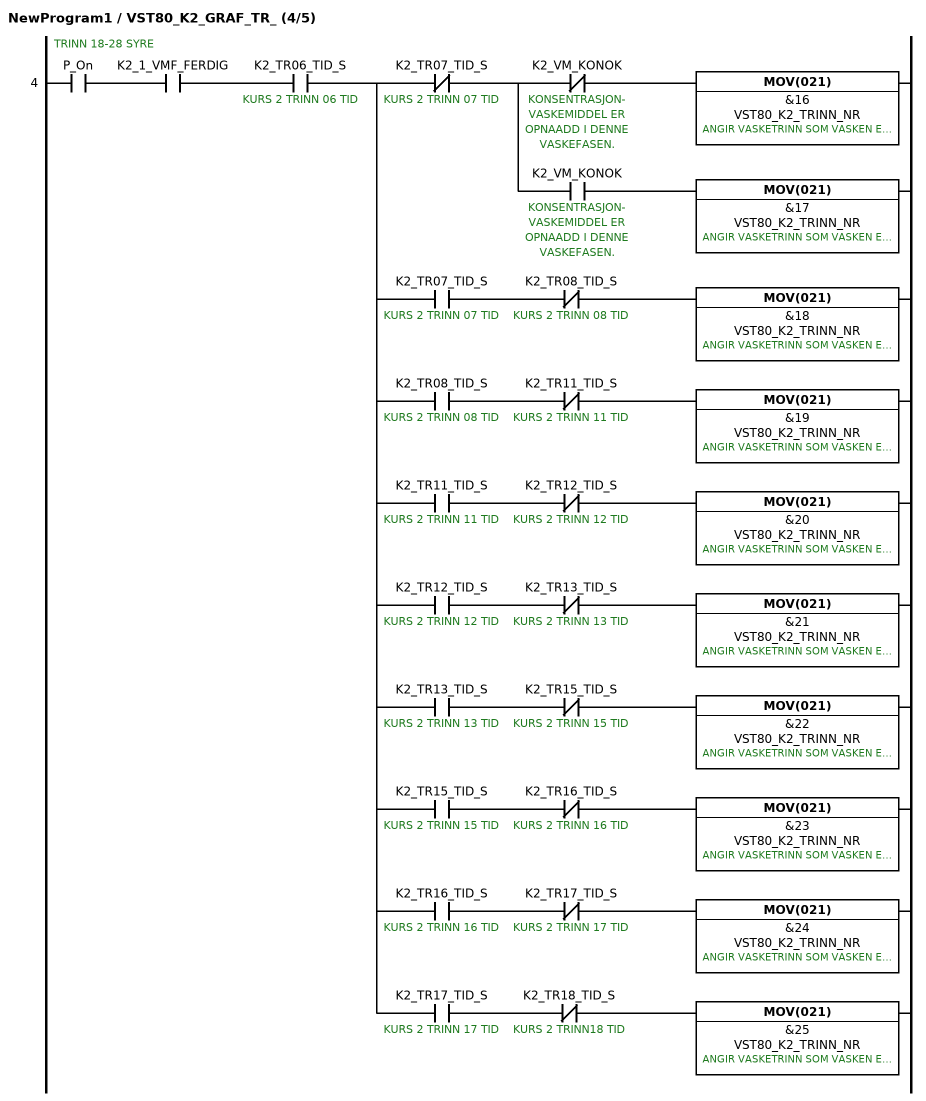
; [picture p264: NewProgram1 / VST80_K2_GRAF_TR_, rungs 4-4]
; rung 4: TRINN 18-28 SYRE
LD P_On
AND K2_1_VMF_FERDIG
AND K2_TR06_TID_S  ; KURS 2 TRINN 06 TID
OUT TR0
ANDNOT K2_TR07_TID_S  ; KURS 2 TRINN 07 TID
OUT TR1
ANDNOT K2_VM_KONOK  ; KONSENTRASJON-VASKEMIDDEL ER OPNAADD I DENNE VASKEFASEN.
MOV(021) &16 VST80_K2_TRINN_NR  ; ANGIR VASKETRINN SOM VASKEN ER I
LD TR1
AND K2_VM_KONOK  ; KONSENTRASJON-VASKEMIDDEL ER OPNAADD I DENNE VASKEFASEN.
MOV(021) &17 VST80_K2_TRINN_NR  ; ANGIR VASKETRINN SOM VASKEN ER I
LD TR0
AND K2_TR07_TID_S  ; KURS 2 TRINN 07 TID
ANDNOT K2_TR08_TID_S  ; KURS 2 TRINN 08 TID
MOV(021) &18 VST80_K2_TRINN_NR  ; ANGIR VASKETRINN SOM VASKEN ER I
LD TR0
AND K2_TR08_TID_S  ; KURS 2 TRINN 08 TID
ANDNOT K2_TR11_TID_S  ; KURS 2 TRINN 11 TID
MOV(021) &19 VST80_K2_TRINN_NR  ; ANGIR VASKETRINN SOM VASKEN ER I
LD TR0
AND K2_TR11_TID_S  ; KURS 2 TRINN 11 TID
ANDNOT K2_TR12_TID_S  ; KURS 2 TRINN 12 TID
MOV(021) &20 VST80_K2_TRINN_NR  ; ANGIR VASKETRINN SOM VASKEN ER I
LD TR0
AND K2_TR12_TID_S  ; KURS 2 TRINN 12 TID
ANDNOT K2_TR13_TID_S  ; KURS 2 TRINN 13 TID
MOV(021) &21 VST80_K2_TRINN_NR  ; ANGIR VASKETRINN SOM VASKEN ER I
LD TR0
AND K2_TR13_TID_S  ; KURS 2 TRINN 13 TID
ANDNOT K2_TR15_TID_S  ; KURS 2 TRINN 15 TID
MOV(021) &22 VST80_K2_TRINN_NR  ; ANGIR VASKETRINN SOM VASKEN ER I
LD TR0
AND K2_TR15_TID_S  ; KURS 2 TRINN 15 TID
ANDNOT K2_TR16_TID_S  ; KURS 2 TRINN 16 TID
MOV(021) &23 VST80_K2_TRINN_NR  ; ANGIR VASKETRINN SOM VASKEN ER I
LD TR0
AND K2_TR16_TID_S  ; KURS 2 TRINN 16 TID
ANDNOT K2_TR17_TID_S  ; KURS 2 TRINN 17 TID
MOV(021) &24 VST80_K2_TRINN_NR  ; ANGIR VASKETRINN SOM VASKEN ER I
LD TR0
AND K2_TR17_TID_S  ; KURS 2 TRINN 17 TID
ANDNOT K2_TR18_TID_S  ; KURS 2 TRINN18 TID
MOV(021) &25 VST80_K2_TRINN_NR  ; ANGIR VASKETRINN SOM VASKEN ER I

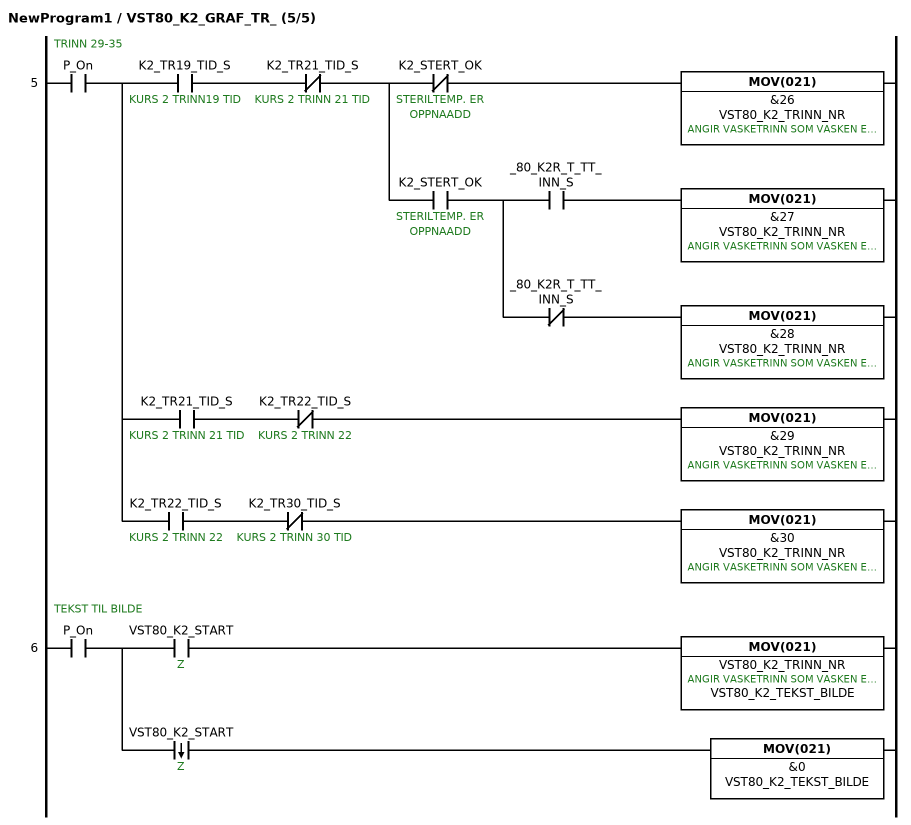
; rung 5: TRINN 29-35
LD P_On
OUT TR0
AND K2_TR19_TID_S  ; KURS 2 TRINN19 TID
ANDNOT K2_TR21_TID_S  ; KURS 2 TRINN 21 TID
OUT TR1
ANDNOT K2_STERT_OK  ; STERILTEMP. ER OPPNAADD
MOV(021) &26 VST80_K2_TRINN_NR  ; ANGIR VASKETRINN SOM VASKEN ER I
LD TR1
AND K2_STERT_OK  ; STERILTEMP. ER OPPNAADD
OUT TR1
AND _80_K2R_T_TT_INN_S
MOV(021) &27 VST80_K2_TRINN_NR  ; ANGIR VASKETRINN SOM VASKEN ER I
LD TR1
ANDNOT _80_K2R_T_TT_INN_S
MOV(021) &28 VST80_K2_TRINN_NR  ; ANGIR VASKETRINN SOM VASKEN ER I
LD TR0
AND K2_TR21_TID_S  ; KURS 2 TRINN 21 TID
ANDNOT K2_TR22_TID_S  ; KURS 2 TRINN 22
MOV(021) &29 VST80_K2_TRINN_NR  ; ANGIR VASKETRINN SOM VASKEN ER I
LD TR0
AND K2_TR22_TID_S  ; KURS 2 TRINN 22
ANDNOT K2_TR30_TID_S  ; KURS 2 TRINN 30 TID
MOV(021) &30 VST80_K2_TRINN_NR  ; ANGIR VASKETRINN SOM VASKEN ER I
; rung 6: TEKST TIL BILDE
LD P_On
OUT TR0
AND VST80_K2_START  ; Z
MOV(021) VST80_K2_TRINN_NR VST80_K2_TEKST_BILDE  ; ANGIR VASKETRINN SOM VASKEN ER I
LD TR0
%AND VST80_K2_START  ; Z
MOV(021) &0 VST80_K2_TEKST_BILDE
; rung 7: Ingen_kommentar_funnet

### Section VST80_K2_GRAF_FEIL_TXT

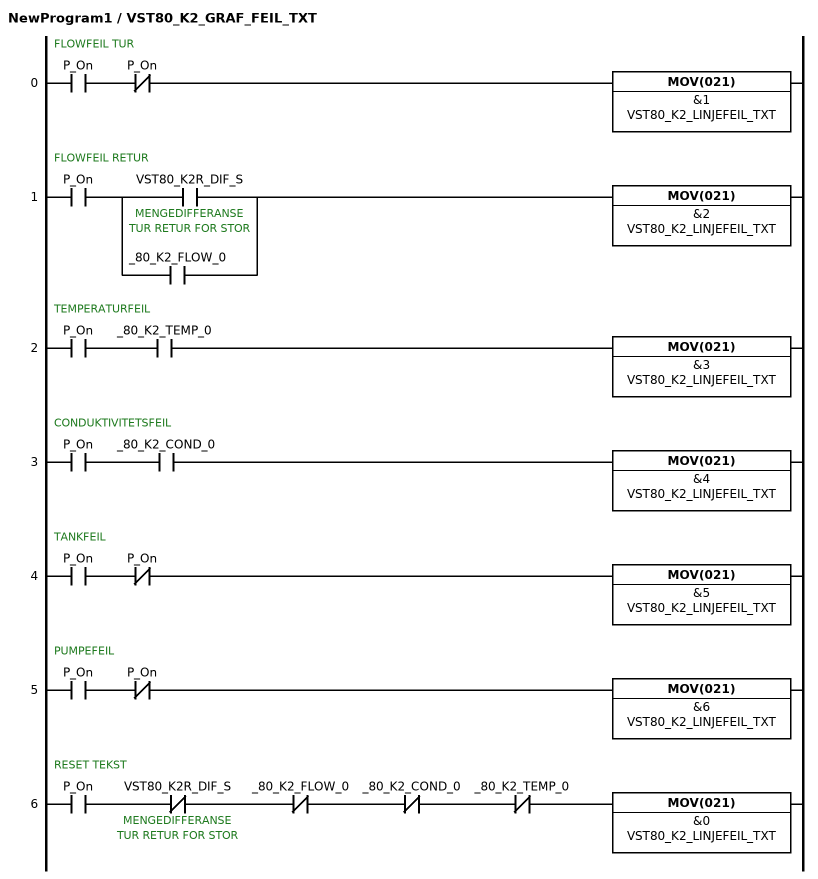
; rung 0: FLOWFEIL TUR
LD P_On
ANDNOT P_On
MOV(021) &1 VST80_K2_LINJEFEIL_TXT
; rung 1: FLOWFEIL RETUR
LD P_On
LD VST80_K2R_DIF_S  ; MENGEDIFFERANSE TUR RETUR FOR STOR
OR _80_K2_FLOW_0
ANDLD
MOV(021) &2 VST80_K2_LINJEFEIL_TXT
; rung 2: TEMPERATURFEIL
LD P_On
AND _80_K2_TEMP_0
MOV(021) &3 VST80_K2_LINJEFEIL_TXT
; rung 3: CONDUKTIVITETSFEIL
LD P_On
AND _80_K2_COND_0
MOV(021) &4 VST80_K2_LINJEFEIL_TXT
; rung 4: TANKFEIL
LD P_On
ANDNOT P_On
MOV(021) &5 VST80_K2_LINJEFEIL_TXT
; rung 5: PUMPEFEIL
LD P_On
ANDNOT P_On
MOV(021) &6 VST80_K2_LINJEFEIL_TXT
; rung 6: RESET TEKST
LD P_On
ANDNOT VST80_K2R_DIF_S  ; MENGEDIFFERANSE TUR RETUR FOR STOR
ANDNOT _80_K2_FLOW_0
ANDNOT _80_K2_COND_0
ANDNOT _80_K2_TEMP_0
MOV(021) &0 VST80_K2_LINJEFEIL_TXT
; rung 7: Ingen_kommentar_funnet

### Section VST80_K2_MENGDE_FASESKIFTE

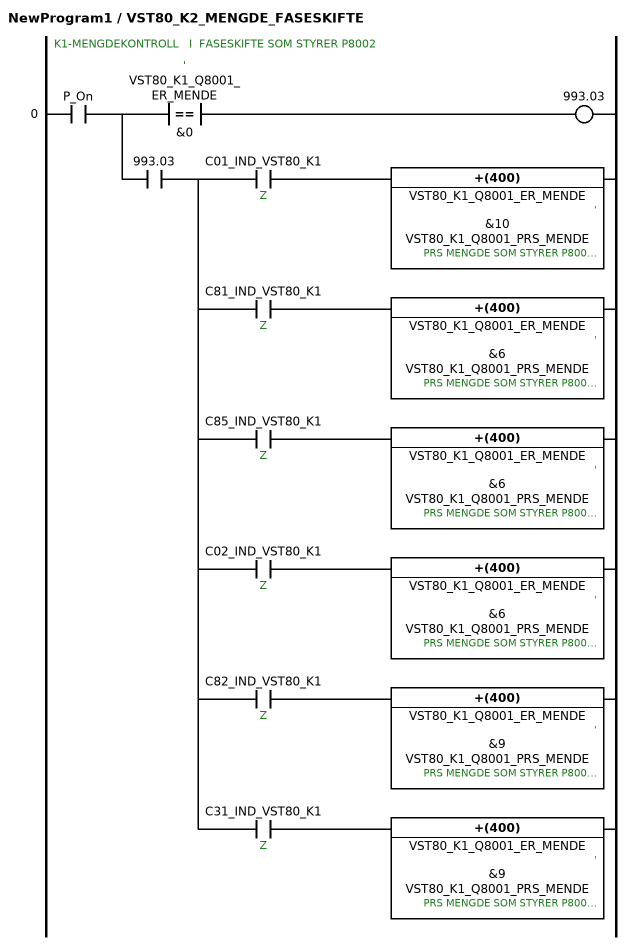
; rung 0: K1-MENGDEKONTROLL   I  FASESKIFTE SOM STYRER P8002
LD P_On
OUT TR0
AND=(300) VST80_K1_Q8001_ER_MENDE &0  ; '
OUT 993.03
LD TR0
AND 993.03
OUT TR0
AND C01_IND_VST80_K1  ; Z
+(400) VST80_K1_Q8001_ER_MENDE &10 VST80_K1_Q8001_PRS_MENDE  ; ', PRS MENGDE SOM STYRER P8001 VED FASESKIFTE
LD TR0
AND C81_IND_VST80_K1  ; Z
+(400) VST80_K1_Q8001_ER_MENDE &6 VST80_K1_Q8001_PRS_MENDE  ; ', PRS MENGDE SOM STYRER P8001 VED FASESKIFTE
LD TR0
AND C85_IND_VST80_K1  ; Z
+(400) VST80_K1_Q8001_ER_MENDE &6 VST80_K1_Q8001_PRS_MENDE  ; ', PRS MENGDE SOM STYRER P8001 VED FASESKIFTE
LD TR0
AND C02_IND_VST80_K1  ; Z
+(400) VST80_K1_Q8001_ER_MENDE &6 VST80_K1_Q8001_PRS_MENDE  ; ', PRS MENGDE SOM STYRER P8001 VED FASESKIFTE
LD TR0
AND C82_IND_VST80_K1  ; Z
+(400) VST80_K1_Q8001_ER_MENDE &9 VST80_K1_Q8001_PRS_MENDE  ; ', PRS MENGDE SOM STYRER P8001 VED FASESKIFTE
LD TR0
AND C31_IND_VST80_K1  ; Z
+(400) VST80_K1_Q8001_ER_MENDE &9 VST80_K1_Q8001_PRS_MENDE  ; ', PRS MENGDE SOM STYRER P8001 VED FASESKIFTE
; rung 1: Ingen_kommentar_funnet

### Section VST80_K2_TR_VEKS
; VST80 KURS2 VEKSLING AV TRINN.

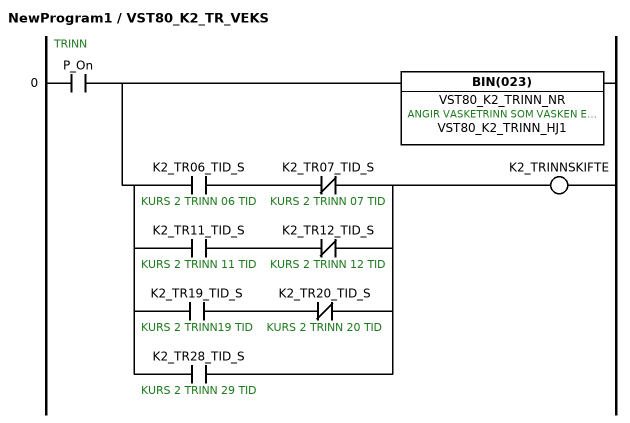
; rung 0: TRINN
LD P_On
BIN(023) VST80_K2_TRINN_NR VST80_K2_TRINN_HJ1  ; ANGIR VASKETRINN SOM VASKEN ER I
LD K2_TR06_TID_S  ; KURS 2 TRINN 06 TID
ANDNOT K2_TR07_TID_S  ; KURS 2 TRINN 07 TID
LD K2_TR11_TID_S  ; KURS 2 TRINN 11 TID
ANDNOT K2_TR12_TID_S  ; KURS 2 TRINN 12 TID
ORLD
LD K2_TR19_TID_S  ; KURS 2 TRINN19 TID
ANDNOT K2_TR20_TID_S  ; KURS 2 TRINN 20 TID
ORLD
OR K2_TR28_TID_S  ; KURS 2 TRINN 29 TID
ANDLD
OUT K2_TRINNSKIFTE
; rung 1: Ingen_kommentar_funnet

### Section V80_K2_FEIL_RET
; FEIL I RETUR / FLOW / TEMP / COND

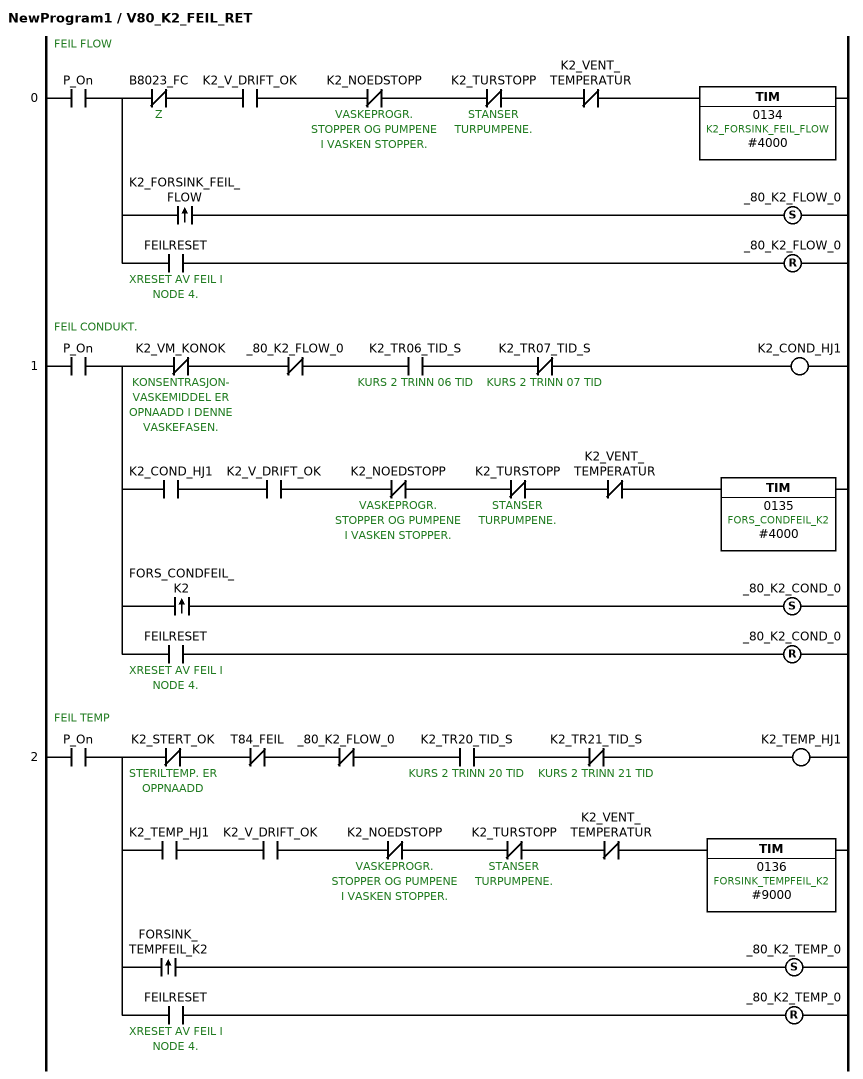
; rung 0: FEIL FLOW
LD P_On
OUT TR0
ANDNOT B8023_FC  ; Z
AND K2_V_DRIFT_OK
ANDNOT K2_NOEDSTOPP  ; VASKEPROGR. STOPPER OG PUMPENE I VASKEN STOPPER.
ANDNOT K2_TURSTOPP  ; STANSER TURPUMPENE.
ANDNOT K2_VENT_TEMPERATUR
TIM 0134 #4000  ; K2_FORSINK_FEIL_FLOW
LD TR0
@AND K2_FORSINK_FEIL_FLOW
SET _80_K2_FLOW_0
LD TR0
AND FEILRESET  ; XRESET AV FEIL I NODE 4.
RSET _80_K2_FLOW_0
; rung 1: FEIL CONDUKT.
LD P_On
OUT TR0
ANDNOT K2_VM_KONOK  ; KONSENTRASJON-VASKEMIDDEL ER OPNAADD I DENNE VASKEFASEN.
ANDNOT _80_K2_FLOW_0
AND K2_TR06_TID_S  ; KURS 2 TRINN 06 TID
ANDNOT K2_TR07_TID_S  ; KURS 2 TRINN 07 TID
OUT K2_COND_HJ1
LD TR0
AND K2_COND_HJ1
AND K2_V_DRIFT_OK
ANDNOT K2_NOEDSTOPP  ; VASKEPROGR. STOPPER OG PUMPENE I VASKEN STOPPER.
ANDNOT K2_TURSTOPP  ; STANSER TURPUMPENE.
ANDNOT K2_VENT_TEMPERATUR
TIM 0135 #4000  ; FORS_CONDFEIL_K2
LD TR0
@AND FORS_CONDFEIL_K2
SET _80_K2_COND_0
LD TR0
AND FEILRESET  ; XRESET AV FEIL I NODE 4.
RSET _80_K2_COND_0
; rung 2: FEIL TEMP
LD P_On
OUT TR0
ANDNOT K2_STERT_OK  ; STERILTEMP. ER OPPNAADD
ANDNOT T84_FEIL
ANDNOT _80_K2_FLOW_0
AND K2_TR20_TID_S  ; KURS 2 TRINN 20 TID
ANDNOT K2_TR21_TID_S  ; KURS 2 TRINN 21 TID
OUT K2_TEMP_HJ1
LD TR0
AND K2_TEMP_HJ1
AND K2_V_DRIFT_OK
ANDNOT K2_NOEDSTOPP  ; VASKEPROGR. STOPPER OG PUMPENE I VASKEN STOPPER.
ANDNOT K2_TURSTOPP  ; STANSER TURPUMPENE.
ANDNOT K2_VENT_TEMPERATUR
TIM 0136 #9000  ; FORSINK_TEMPFEIL_K2
LD TR0
@AND FORSINK_TEMPFEIL_K2
SET _80_K2_TEMP_0
LD TR0
AND FEILRESET  ; XRESET AV FEIL I NODE 4.
RSET _80_K2_TEMP_0
; rung 3: Ingen_kommentar_funnet

### Section VST80_K2_VASKERAPPORT
; VST80 / KURS1 VASKERAPPORT

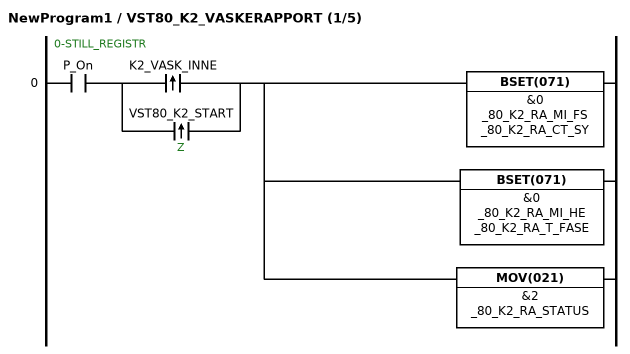
; rung 0: 0-STILL_REGISTR
LD P_On
@LD K2_VASK_INNE
@OR VST80_K2_START  ; Z
ANDLD
BSET(071) &0 _80_K2_RA_MI_FS _80_K2_RA_CT_SY
BSET(071) &0 _80_K2_RA_MI_HE _80_K2_RA_T_FASE
MOV(021) &2 _80_K2_RA_STATUS

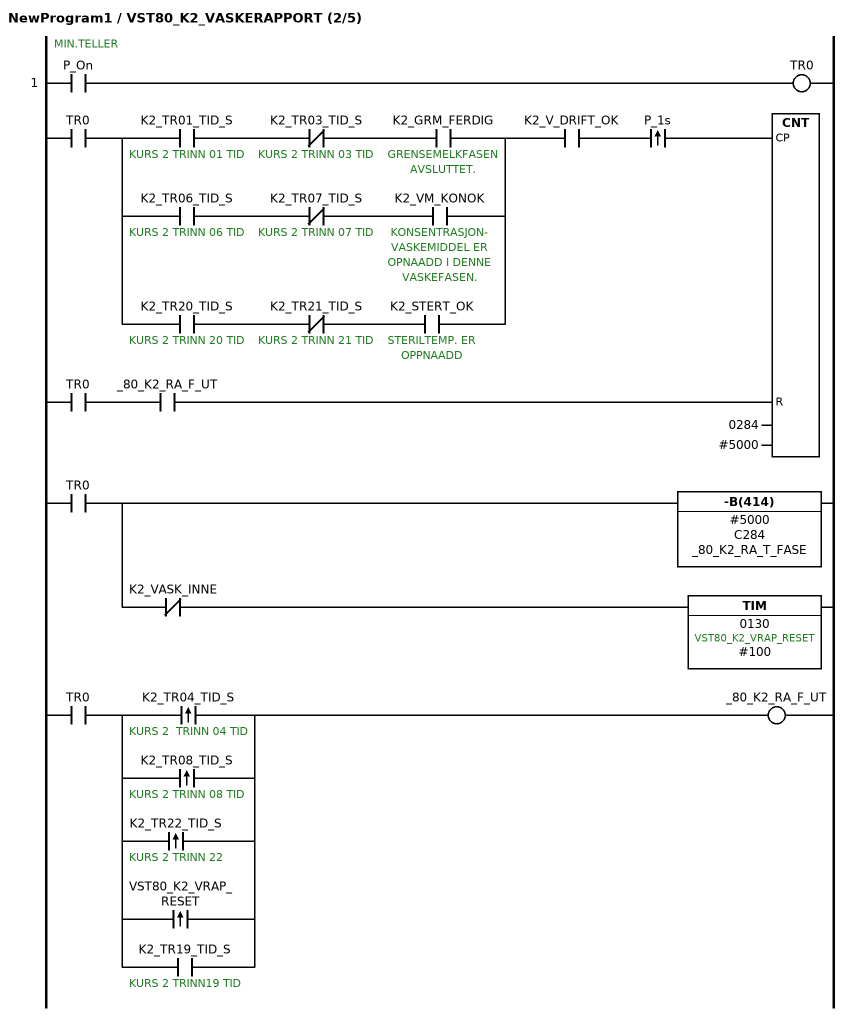
; rung 1: MIN.TELLER
LD P_On
OUT TR0
LD K2_TR01_TID_S  ; KURS 2 TRINN 01 TID
ANDNOT K2_TR03_TID_S  ; KURS 2 TRINN 03 TID
AND K2_GRM_FERDIG  ; GRENSEMELKFASEN AVSLUTTET.
LD K2_TR06_TID_S  ; KURS 2 TRINN 06 TID
ANDNOT K2_TR07_TID_S  ; KURS 2 TRINN 07 TID
AND K2_VM_KONOK  ; KONSENTRASJON-VASKEMIDDEL ER OPNAADD I DENNE VASKEFASEN.
ORLD
LD K2_TR20_TID_S  ; KURS 2 TRINN 20 TID
ANDNOT K2_TR21_TID_S  ; KURS 2 TRINN 21 TID
AND K2_STERT_OK  ; STERILTEMP. ER OPPNAADD
ORLD
ANDLD
AND K2_V_DRIFT_OK
@AND P_1s
LD TR0
AND _80_K2_RA_F_UT
CNT 0284 #5000
LD TR0
-B(414) #5000 C284 _80_K2_RA_T_FASE
ANDNOT K2_VASK_INNE
TIM 0130 #100  ; VST80_K2_VRAP_RESET
LD TR0
@LD K2_TR04_TID_S  ; KURS 2  TRINN 04 TID
@OR K2_TR08_TID_S  ; KURS 2 TRINN 08 TID
@OR K2_TR22_TID_S  ; KURS 2 TRINN 22
@OR VST80_K2_VRAP_RESET
OR K2_TR19_TID_S  ; KURS 2 TRINN19 TID
ANDLD
OUT _80_K2_RA_F_UT

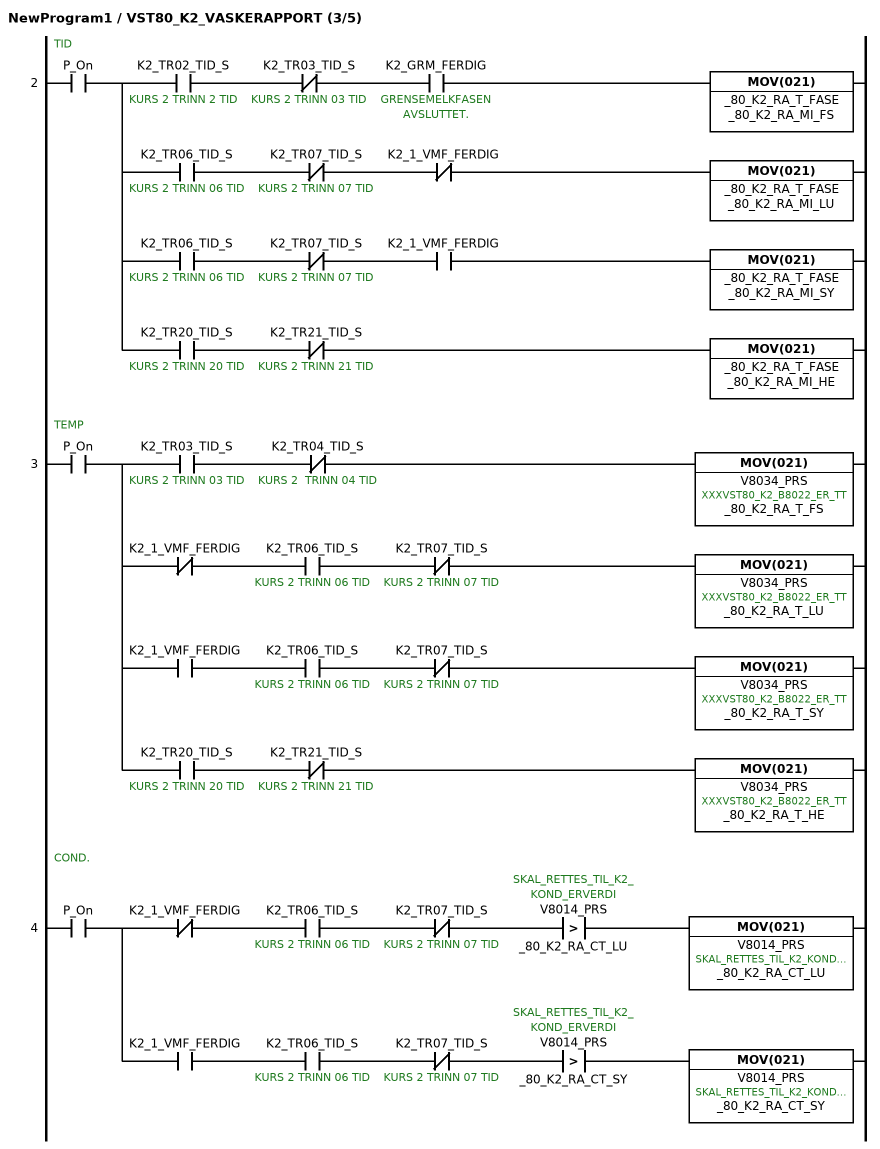
; rung 2: TID
LD P_On
OUT TR0
AND K2_TR02_TID_S  ; KURS 2 TRINN 2 TID
ANDNOT K2_TR03_TID_S  ; KURS 2 TRINN 03 TID
AND K2_GRM_FERDIG  ; GRENSEMELKFASEN AVSLUTTET.
MOV(021) _80_K2_RA_T_FASE _80_K2_RA_MI_FS
LD TR0
AND K2_TR06_TID_S  ; KURS 2 TRINN 06 TID
ANDNOT K2_TR07_TID_S  ; KURS 2 TRINN 07 TID
ANDNOT K2_1_VMF_FERDIG
MOV(021) _80_K2_RA_T_FASE _80_K2_RA_MI_LU
LD TR0
AND K2_TR06_TID_S  ; KURS 2 TRINN 06 TID
ANDNOT K2_TR07_TID_S  ; KURS 2 TRINN 07 TID
AND K2_1_VMF_FERDIG
MOV(021) _80_K2_RA_T_FASE _80_K2_RA_MI_SY
LD TR0
AND K2_TR20_TID_S  ; KURS 2 TRINN 20 TID
ANDNOT K2_TR21_TID_S  ; KURS 2 TRINN 21 TID
MOV(021) _80_K2_RA_T_FASE _80_K2_RA_MI_HE
; rung 3: TEMP
LD P_On
OUT TR0
AND K2_TR03_TID_S  ; KURS 2 TRINN 03 TID
ANDNOT K2_TR04_TID_S  ; KURS 2  TRINN 04 TID
MOV(021) V8034_PRS _80_K2_RA_T_FS  ; XXXVST80_K2_B8022_ER_TT
LD TR0
ANDNOT K2_1_VMF_FERDIG
AND K2_TR06_TID_S  ; KURS 2 TRINN 06 TID
ANDNOT K2_TR07_TID_S  ; KURS 2 TRINN 07 TID
MOV(021) V8034_PRS _80_K2_RA_T_LU  ; XXXVST80_K2_B8022_ER_TT
LD TR0
AND K2_1_VMF_FERDIG
AND K2_TR06_TID_S  ; KURS 2 TRINN 06 TID
ANDNOT K2_TR07_TID_S  ; KURS 2 TRINN 07 TID
MOV(021) V8034_PRS _80_K2_RA_T_SY  ; XXXVST80_K2_B8022_ER_TT
LD TR0
AND K2_TR20_TID_S  ; KURS 2 TRINN 20 TID
ANDNOT K2_TR21_TID_S  ; KURS 2 TRINN 21 TID
MOV(021) V8034_PRS _80_K2_RA_T_HE  ; XXXVST80_K2_B8022_ER_TT
; rung 4: COND.
LD P_On
OUT TR0
ANDNOT K2_1_VMF_FERDIG
AND K2_TR06_TID_S  ; KURS 2 TRINN 06 TID
ANDNOT K2_TR07_TID_S  ; KURS 2 TRINN 07 TID
AND>(320) V8014_PRS _80_K2_RA_CT_LU  ; SKAL_RETTES_TIL_K2_KOND_ERVERDI
MOV(021) V8014_PRS _80_K2_RA_CT_LU  ; SKAL_RETTES_TIL_K2_KOND_ERVERDI
LD TR0
AND K2_1_VMF_FERDIG
AND K2_TR06_TID_S  ; KURS 2 TRINN 06 TID
ANDNOT K2_TR07_TID_S  ; KURS 2 TRINN 07 TID
AND>(320) V8014_PRS _80_K2_RA_CT_SY  ; SKAL_RETTES_TIL_K2_KOND_ERVERDI
MOV(021) V8014_PRS _80_K2_RA_CT_SY  ; SKAL_RETTES_TIL_K2_KOND_ERVERDI

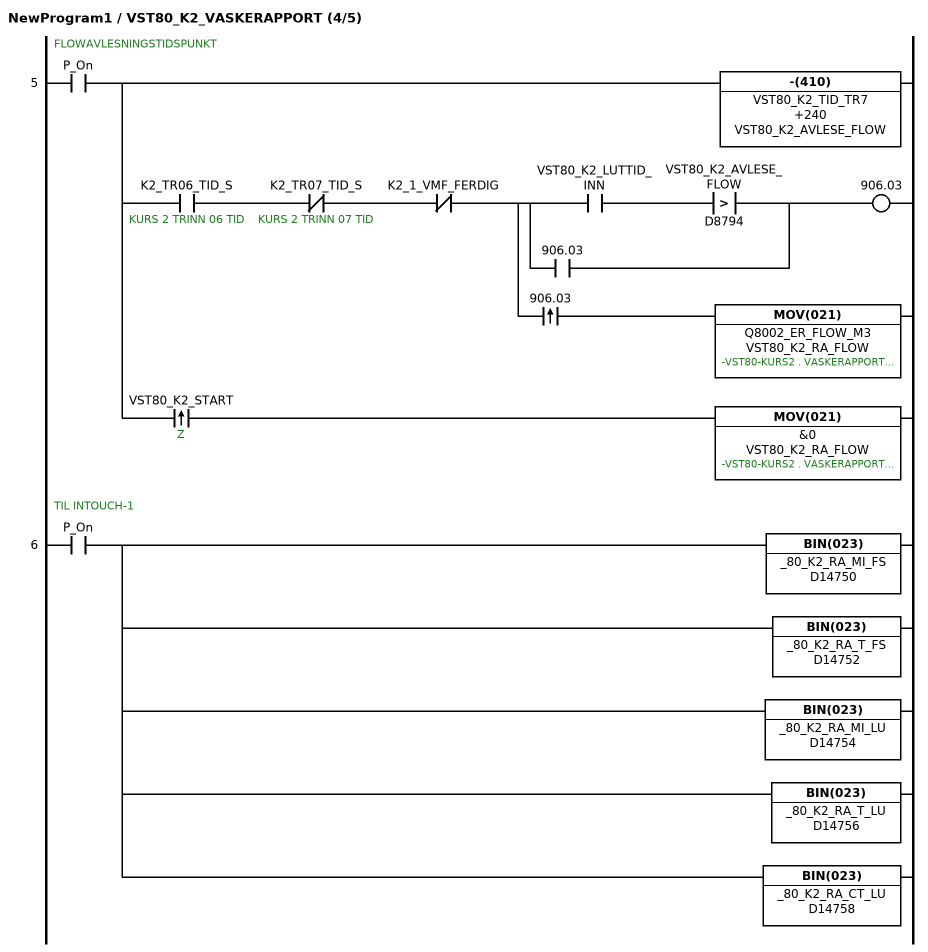
; rung 5: FLOWAVLESNINGSTIDSPUNKT
LD P_On
OUT TR0
-(410) VST80_K2_TID_TR7 +240 VST80_K2_AVLESE_FLOW
AND K2_TR06_TID_S  ; KURS 2 TRINN 06 TID
ANDNOT K2_TR07_TID_S  ; KURS 2 TRINN 07 TID
ANDNOT K2_1_VMF_FERDIG
OUT TR1
LD VST80_K2_LUTTID_INN
AND>(320) VST80_K2_AVLESE_FLOW D8794
OR 906.03
ANDLD
OUT 906.03
LD TR1
@AND 906.03
MOV(021) Q8002_ER_FLOW_M3 VST80_K2_RA_FLOW  ; -VST80-KURS2 . VASKERAPPORT.  FLOW
LD TR0
@AND VST80_K2_START  ; Z
MOV(021) &0 VST80_K2_RA_FLOW  ; -VST80-KURS2 . VASKERAPPORT.  FLOW
; rung 6: TIL INTOUCH-1
LD P_On
BIN(023) _80_K2_RA_MI_FS D14750
BIN(023) _80_K2_RA_T_FS D14752
BIN(023) _80_K2_RA_MI_LU D14754
BIN(023) _80_K2_RA_T_LU D14756
BIN(023) _80_K2_RA_CT_LU D14758

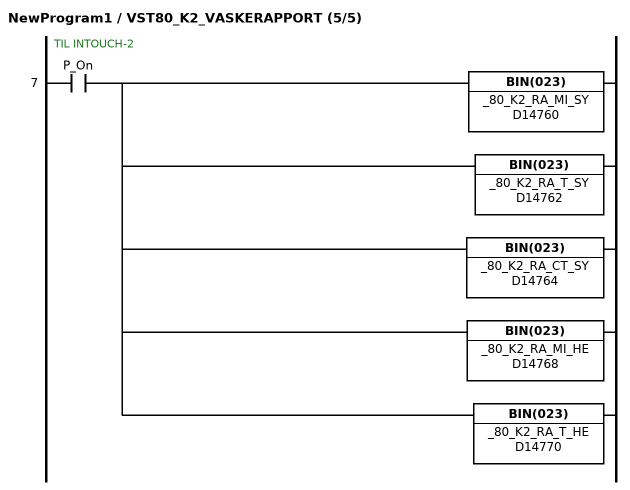
; rung 7: TIL INTOUCH-2
LD P_On
BIN(023) _80_K2_RA_MI_SY D14760
BIN(023) _80_K2_RA_T_SY D14762
BIN(023) _80_K2_RA_CT_SY D14764
BIN(023) _80_K2_RA_MI_HE D14768
BIN(023) _80_K2_RA_T_HE D14770
; rung 8: Ingen_kommentar_funnet

### Section VST80_K2_REGULATORER

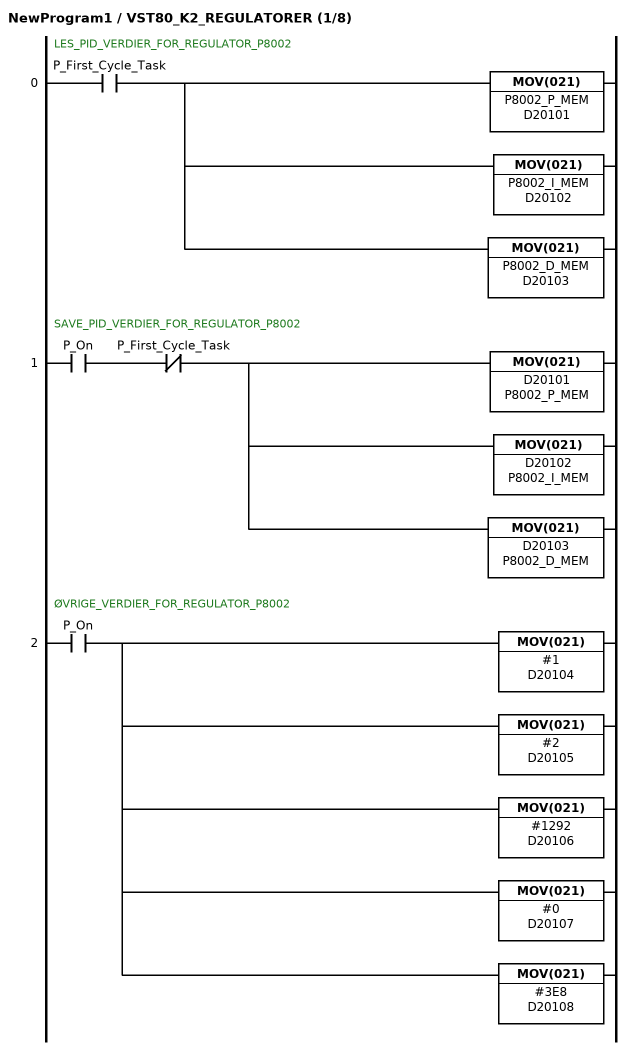
; rung 0: LES_PID_VERDIER_FOR_REGULATOR_P8002
LD P_First_Cycle_Task
MOV(021) P8002_P_MEM D20101
MOV(021) P8002_I_MEM D20102
MOV(021) P8002_D_MEM D20103
; rung 1: SAVE_PID_VERDIER_FOR_REGULATOR_P8002
LD P_On
ANDNOT P_First_Cycle_Task
MOV(021) D20101 P8002_P_MEM
MOV(021) D20102 P8002_I_MEM
MOV(021) D20103 P8002_D_MEM
; rung 2: ØVRIGE_VERDIER_FOR_REGULATOR_P8002
LD P_On
MOV(021) #1 D20104
MOV(021) #2 D20105
MOV(021) #1292 D20106
MOV(021) #0 D20107
MOV(021) #3E8 D20108

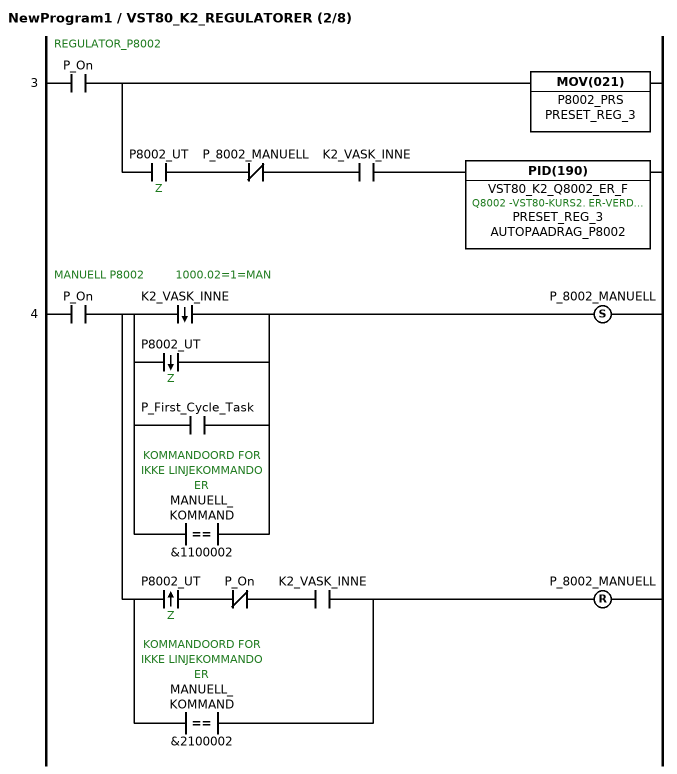
; rung 3: REGULATOR_P8002
LD P_On
MOV(021) P8002_PRS PRESET_REG_3
AND P8002_UT  ; Z
ANDNOT P_8002_MANUELL
AND K2_VASK_INNE
PID(190) VST80_K2_Q8002_ER_F PRESET_REG_3 AUTOPAADRAG_P8002  ; Q8002 -VST80-KURS2. ER-VERDI FLOW I TUR
; rung 4: MANUELL P8002         1000.02=1=MAN
LD P_On
OUT TR0
%LD K2_VASK_INNE
%OR P8002_UT  ; Z
OR P_First_Cycle_Task
OR=L(301) MANUELL_KOMMAND &1100002  ; KOMMANDOORD FOR IKKE LINJEKOMMANDOER
ANDLD
SET P_8002_MANUELL
LD TR0
@LD P8002_UT  ; Z
ANDNOT P_On
AND K2_VASK_INNE
OR=L(301) MANUELL_KOMMAND &2100002  ; KOMMANDOORD FOR IKKE LINJEKOMMANDOER
ANDLD
RSET P_8002_MANUELL

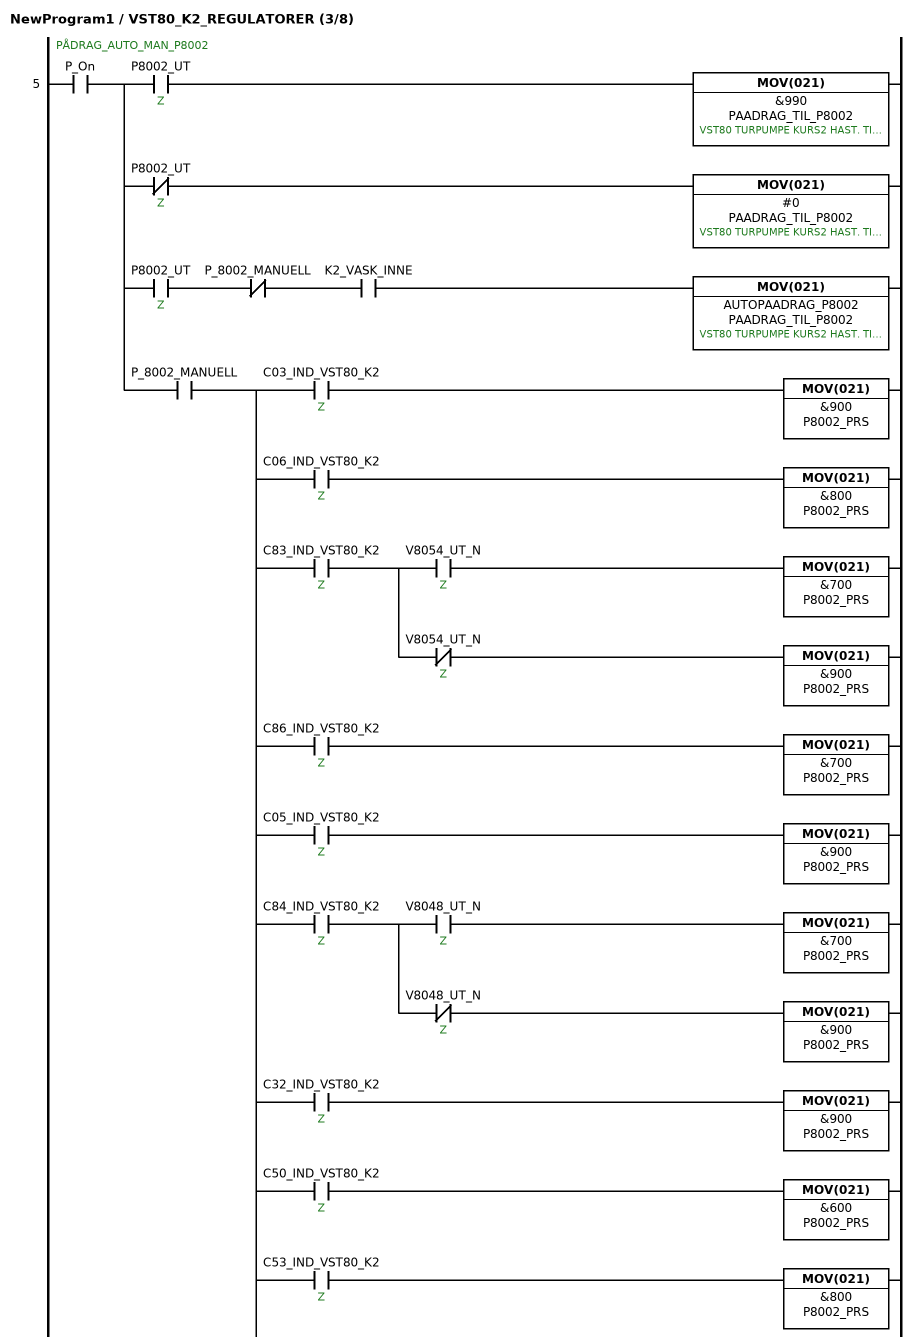

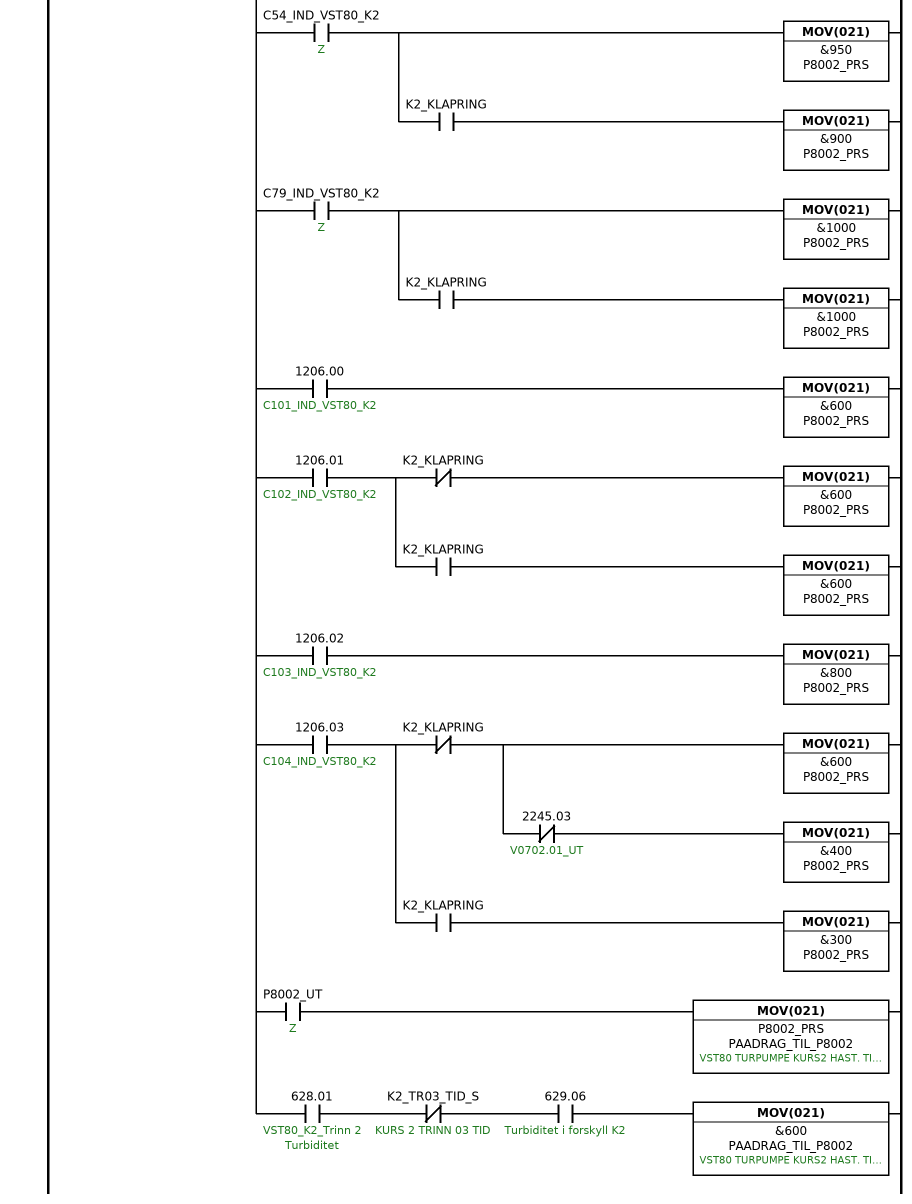
; rung 5: PÅDRAG_AUTO_MAN_P8002
LD P_On
OUT TR0
AND P8002_UT  ; Z
MOV(021) &990 PAADRAG_TIL_P8002  ; VST80 TURPUMPE KURS2 HAST. TIL FR.OMF. P8002
LD TR0
ANDNOT P8002_UT  ; Z
MOV(021) #0 PAADRAG_TIL_P8002  ; VST80 TURPUMPE KURS2 HAST. TIL FR.OMF. P8002
LD TR0
AND P8002_UT  ; Z
ANDNOT P_8002_MANUELL
AND K2_VASK_INNE
MOV(021) AUTOPAADRAG_P8002 PAADRAG_TIL_P8002  ; VST80 TURPUMPE KURS2 HAST. TIL FR.OMF. P8002
LD TR0
AND P_8002_MANUELL
OUT TR0
AND C03_IND_VST80_K2  ; Z
MOV(021) &900 P8002_PRS
LD TR0
AND C06_IND_VST80_K2  ; Z
MOV(021) &800 P8002_PRS
LD TR0
AND C83_IND_VST80_K2  ; Z
OUT TR1
AND V8054_UT_N  ; Z
MOV(021) &700 P8002_PRS
LD TR1
ANDNOT V8054_UT_N  ; Z
MOV(021) &900 P8002_PRS
LD TR0
AND C86_IND_VST80_K2  ; Z
MOV(021) &700 P8002_PRS
LD TR0
AND C05_IND_VST80_K2  ; Z
MOV(021) &900 P8002_PRS
LD TR0
AND C84_IND_VST80_K2  ; Z
OUT TR1
AND V8048_UT_N  ; Z
MOV(021) &700 P8002_PRS
LD TR1
ANDNOT V8048_UT_N  ; Z
MOV(021) &900 P8002_PRS
LD TR0
AND C32_IND_VST80_K2  ; Z
MOV(021) &900 P8002_PRS
LD TR0
AND C50_IND_VST80_K2  ; Z
MOV(021) &600 P8002_PRS
LD TR0
AND C53_IND_VST80_K2  ; Z
MOV(021) &800 P8002_PRS
LD TR0
AND C54_IND_VST80_K2  ; Z
MOV(021) &950 P8002_PRS
AND K2_KLAPRING
MOV(021) &900 P8002_PRS
LD TR0
AND C79_IND_VST80_K2  ; Z
MOV(021) &1000 P8002_PRS
AND K2_KLAPRING
MOV(021) &1000 P8002_PRS
LD TR0
AND 1206.00  ; C101_IND_VST80_K2
MOV(021) &600 P8002_PRS
LD TR0
AND 1206.01  ; C102_IND_VST80_K2
OUT TR1
ANDNOT K2_KLAPRING
MOV(021) &600 P8002_PRS
LD TR1
AND K2_KLAPRING
MOV(021) &600 P8002_PRS
LD TR0
AND 1206.02  ; C103_IND_VST80_K2
MOV(021) &800 P8002_PRS
LD TR0
AND 1206.03  ; C104_IND_VST80_K2
OUT TR1
ANDNOT K2_KLAPRING
MOV(021) &600 P8002_PRS
ANDNOT 2245.03  ; V0702.01_UT
MOV(021) &400 P8002_PRS
LD TR1
AND K2_KLAPRING
MOV(021) &300 P8002_PRS
LD TR0
AND P8002_UT  ; Z
MOV(021) P8002_PRS PAADRAG_TIL_P8002  ; VST80 TURPUMPE KURS2 HAST. TIL FR.OMF. P8002
LD TR0
AND 628.01  ; VST80_K2_Trinn 2 Turbiditet
ANDNOT K2_TR03_TID_S  ; KURS 2 TRINN 03 TID
AND 629.06  ; Turbiditet i forskyll K2
MOV(021) &600 PAADRAG_TIL_P8002  ; VST80 TURPUMPE KURS2 HAST. TIL FR.OMF. P8002

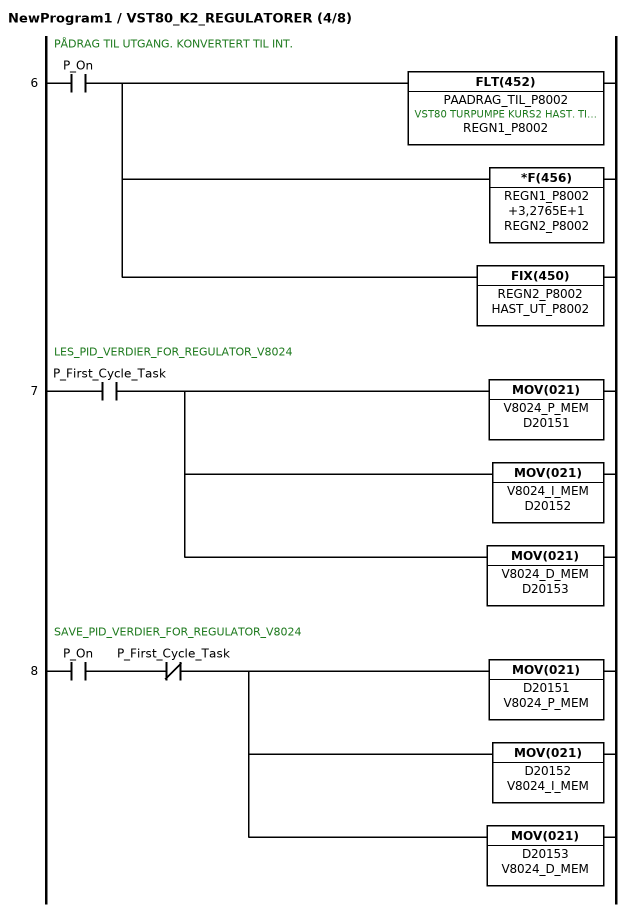
; rung 6: PÅDRAG TIL UTGANG. KONVERTERT TIL INT.
LD P_On
FLT(452) PAADRAG_TIL_P8002 REGN1_P8002  ; VST80 TURPUMPE KURS2 HAST. TIL FR.OMF. P8002
*F(456) REGN1_P8002 +3,2765E+1 REGN2_P8002
FIX(450) REGN2_P8002 HAST_UT_P8002
; rung 7: LES_PID_VERDIER_FOR_REGULATOR_V8024
LD P_First_Cycle_Task
MOV(021) V8024_P_MEM D20151
MOV(021) V8024_I_MEM D20152
MOV(021) V8024_D_MEM D20153
; rung 8: SAVE_PID_VERDIER_FOR_REGULATOR_V8024
LD P_On
ANDNOT P_First_Cycle_Task
MOV(021) D20151 V8024_P_MEM
MOV(021) D20152 V8024_I_MEM
MOV(021) D20153 V8024_D_MEM

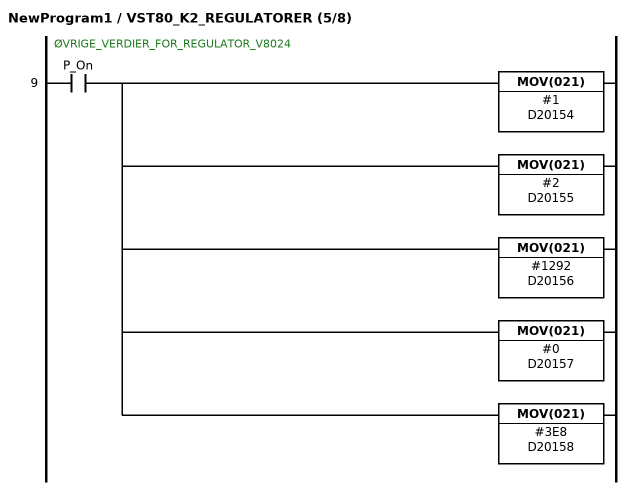
; rung 9: ØVRIGE_VERDIER_FOR_REGULATOR_V8024
LD P_On
MOV(021) #1 D20154
MOV(021) #2 D20155
MOV(021) #1292 D20156
MOV(021) #0 D20157
MOV(021) #3E8 D20158

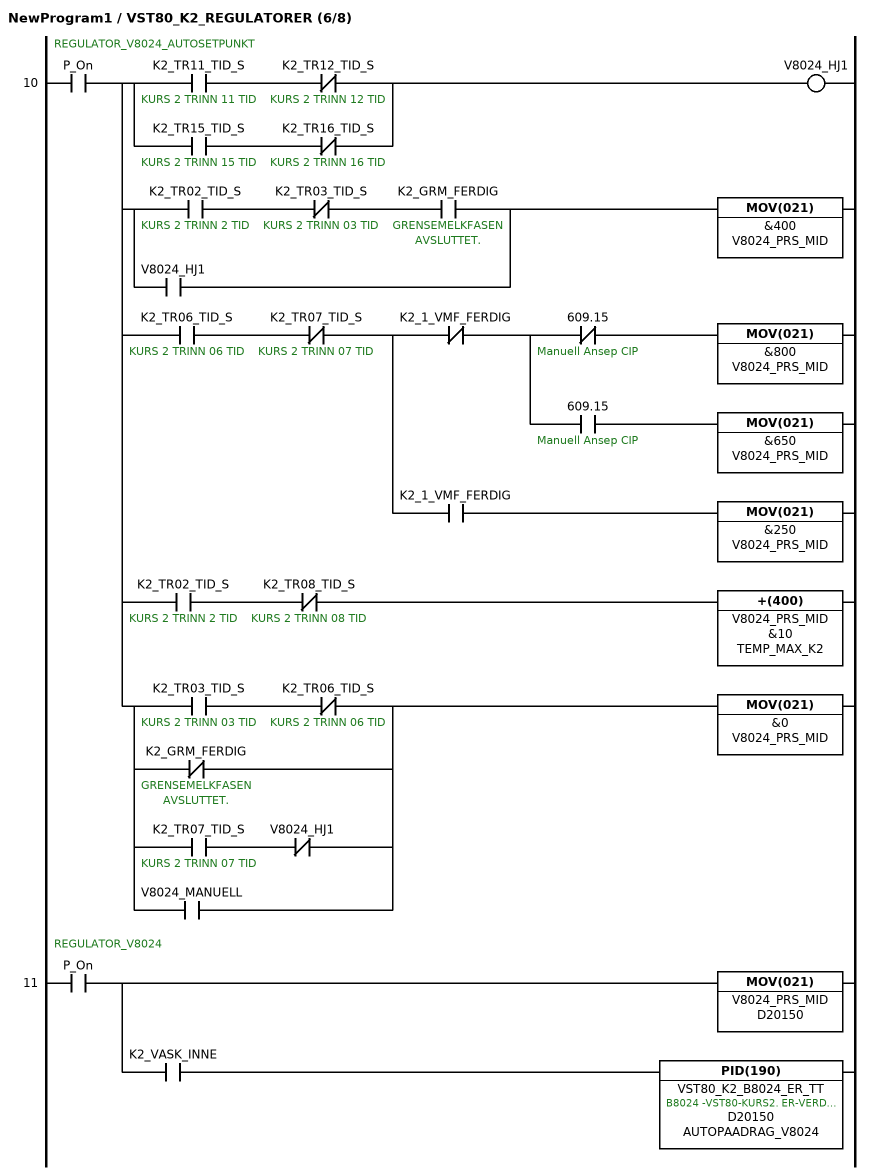
; rung 10: REGULATOR_V8024_AUTOSETPUNKT
LD P_On
OUT TR0
LD K2_TR11_TID_S  ; KURS 2 TRINN 11 TID
ANDNOT K2_TR12_TID_S  ; KURS 2 TRINN 12 TID
LD K2_TR15_TID_S  ; KURS 2 TRINN 15 TID
ANDNOT K2_TR16_TID_S  ; KURS 2 TRINN 16 TID
ORLD
ANDLD
OUT V8024_HJ1
LD TR0
LD K2_TR02_TID_S  ; KURS 2 TRINN 2 TID
ANDNOT K2_TR03_TID_S  ; KURS 2 TRINN 03 TID
AND K2_GRM_FERDIG  ; GRENSEMELKFASEN AVSLUTTET.
OR V8024_HJ1
ANDLD
MOV(021) &400 V8024_PRS_MID
LD TR0
AND K2_TR06_TID_S  ; KURS 2 TRINN 06 TID
ANDNOT K2_TR07_TID_S  ; KURS 2 TRINN 07 TID
OUT TR1
ANDNOT K2_1_VMF_FERDIG
OUT TR2
ANDNOT 609.15  ; Manuell Ansep CIP
MOV(021) &800 V8024_PRS_MID
LD TR2
AND 609.15  ; Manuell Ansep CIP
MOV(021) &650 V8024_PRS_MID
LD TR1
AND K2_1_VMF_FERDIG
MOV(021) &250 V8024_PRS_MID
LD TR0
AND K2_TR02_TID_S  ; KURS 2 TRINN 2 TID
ANDNOT K2_TR08_TID_S  ; KURS 2 TRINN 08 TID
+(400) V8024_PRS_MID &10 TEMP_MAX_K2
LD TR0
LD K2_TR03_TID_S  ; KURS 2 TRINN 03 TID
ANDNOT K2_TR06_TID_S  ; KURS 2 TRINN 06 TID
ORNOT K2_GRM_FERDIG  ; GRENSEMELKFASEN AVSLUTTET.
LD K2_TR07_TID_S  ; KURS 2 TRINN 07 TID
ANDNOT V8024_HJ1
ORLD
OR V8024_MANUELL
ANDLD
MOV(021) &0 V8024_PRS_MID
; rung 11: REGULATOR_V8024
LD P_On
MOV(021) V8024_PRS_MID D20150
AND K2_VASK_INNE
PID(190) VST80_K2_B8024_ER_TT D20150 AUTOPAADRAG_V8024  ; B8024 -VST80-KURS2. ER-VERDI TEMPERATUR I TUR TIL VST

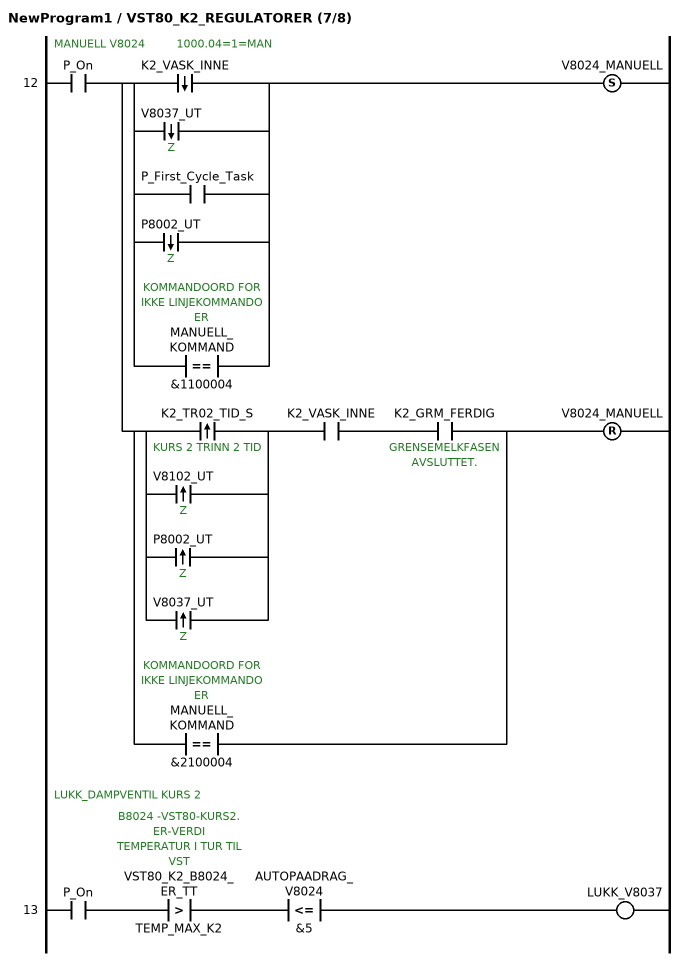
; rung 12: MANUELL V8024         1000.04=1=MAN
LD P_On
OUT TR0
%LD K2_VASK_INNE
%OR V8037_UT  ; Z
OR P_First_Cycle_Task
%OR P8002_UT  ; Z
OR=L(301) MANUELL_KOMMAND &1100004  ; KOMMANDOORD FOR IKKE LINJEKOMMANDOER
ANDLD
SET V8024_MANUELL
LD TR0
@LD K2_TR02_TID_S  ; KURS 2 TRINN 2 TID
@OR V8102_UT  ; Z
@OR P8002_UT  ; Z
@OR V8037_UT  ; Z
AND K2_VASK_INNE
AND K2_GRM_FERDIG  ; GRENSEMELKFASEN AVSLUTTET.
OR=L(301) MANUELL_KOMMAND &2100004  ; KOMMANDOORD FOR IKKE LINJEKOMMANDOER
ANDLD
RSET V8024_MANUELL
; rung 13: LUKK_DAMPVENTIL KURS 2
LD P_On
AND>(320) VST80_K2_B8024_ER_TT TEMP_MAX_K2  ; B8024 -VST80-KURS2. ER-VERDI TEMPERATUR I TUR TIL VST
AND<=(315) AUTOPAADRAG_V8024 &5
OUT LUKK_V8037

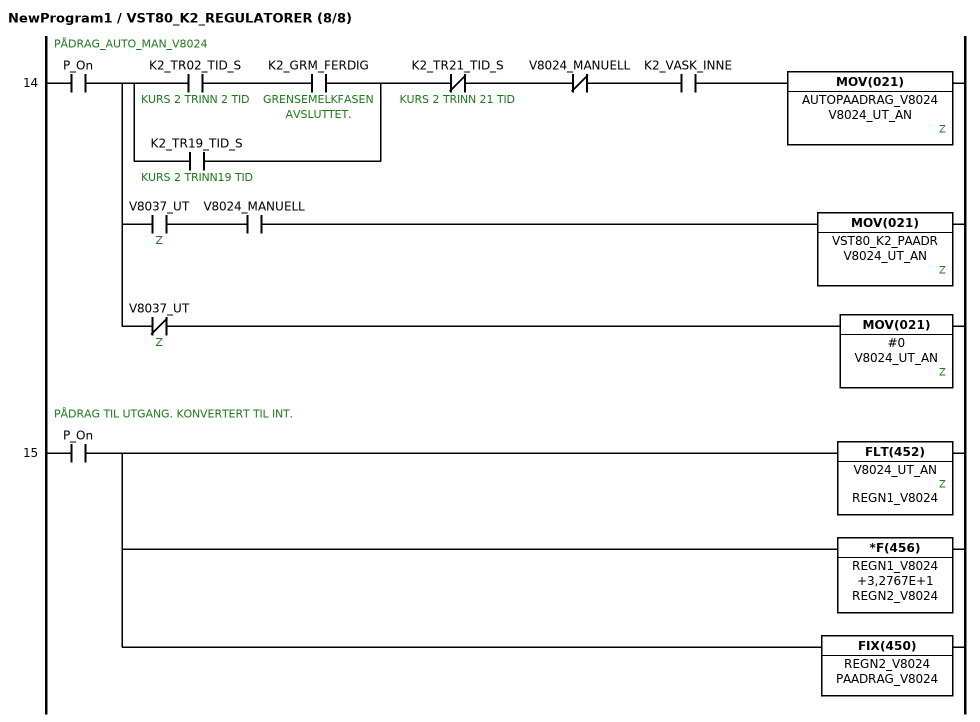
; rung 14: PÅDRAG_AUTO_MAN_V8024
LD P_On
OUT TR0
LD K2_TR02_TID_S  ; KURS 2 TRINN 2 TID
AND K2_GRM_FERDIG  ; GRENSEMELKFASEN AVSLUTTET.
OR K2_TR19_TID_S  ; KURS 2 TRINN19 TID
ANDLD
ANDNOT K2_TR21_TID_S  ; KURS 2 TRINN 21 TID
ANDNOT V8024_MANUELL
AND K2_VASK_INNE
MOV(021) AUTOPAADRAG_V8024 V8024_UT_AN  ; Z
LD TR0
AND V8037_UT  ; Z
AND V8024_MANUELL
MOV(021) VST80_K2_PAADR V8024_UT_AN  ; Z
LD TR0
ANDNOT V8037_UT  ; Z
MOV(021) #0 V8024_UT_AN  ; Z
; rung 15: PÅDRAG TIL UTGANG. KONVERTERT TIL INT.
LD P_On
FLT(452) V8024_UT_AN REGN1_V8024  ; Z
*F(456) REGN1_V8024 +3,2767E+1 REGN2_V8024
FIX(450) REGN2_V8024 PAADRAG_V8024
; rung 16: Ingen_kommentar_funnet

### Section VST80_AUTOVASK_KURS_2

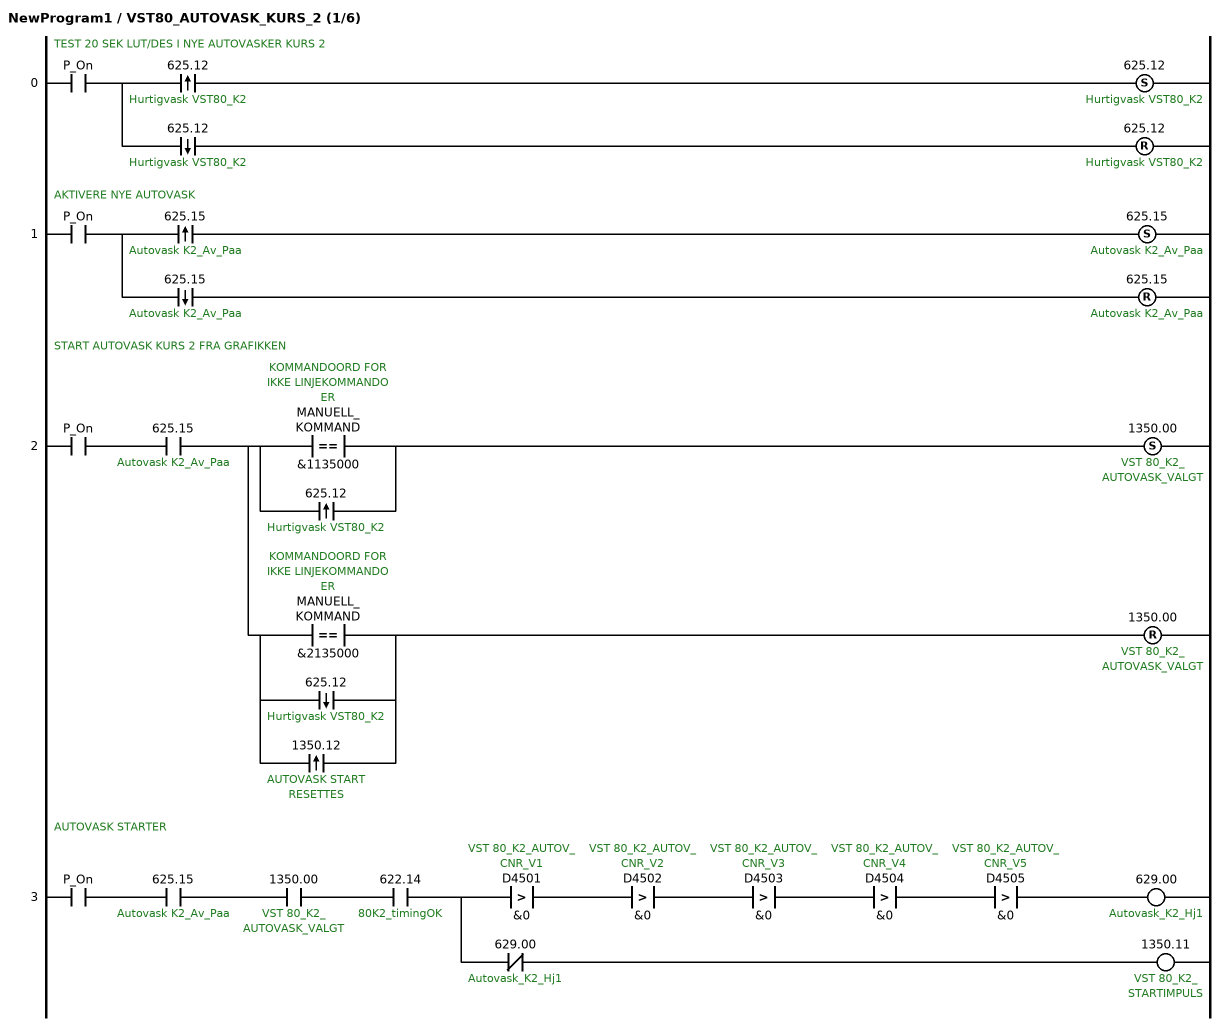
; rung 0: TEST 20 SEK LUT/DES I NYE AUTOVASKER KURS 2
LD P_On
OUT TR0
@AND 625.12  ; Hurtigvask VST80_K2
SET 625.12  ; Hurtigvask VST80_K2
LD TR0
%AND 625.12  ; Hurtigvask VST80_K2
RSET 625.12  ; Hurtigvask VST80_K2
; rung 1: AKTIVERE NYE AUTOVASK
LD P_On
OUT TR0
@AND 625.15  ; Autovask K2_Av_Paa
SET 625.15  ; Autovask K2_Av_Paa
LD TR0
%AND 625.15  ; Autovask K2_Av_Paa
RSET 625.15  ; Autovask K2_Av_Paa
; rung 2: START AUTOVASK KURS 2 FRA GRAFIKKEN
LD P_On
AND 625.15  ; Autovask K2_Av_Paa
OUT TR0
LD=L(301) MANUELL_KOMMAND &1135000  ; KOMMANDOORD FOR IKKE LINJEKOMMANDOER
@OR 625.12  ; Hurtigvask VST80_K2
ANDLD
SET 1350.00  ; VST 80_K2_AUTOVASK_VALGT
LD TR0
LD=L(301) MANUELL_KOMMAND &2135000  ; KOMMANDOORD FOR IKKE LINJEKOMMANDOER
%OR 625.12  ; Hurtigvask VST80_K2
@OR 1350.12  ; AUTOVASK START RESETTES
ANDLD
RSET 1350.00  ; VST 80_K2_AUTOVASK_VALGT
; rung 3: AUTOVASK STARTER
LD P_On
AND 625.15  ; Autovask K2_Av_Paa
AND 1350.00  ; VST 80_K2_AUTOVASK_VALGT
AND 622.14  ; 80K2_timingOK
OUT TR0
AND>(320) D4501 &0  ; VST 80_K2_AUTOV_CNR_V1
AND>(320) D4502 &0  ; VST 80_K2_AUTOV_CNR_V2
AND>(320) D4503 &0  ; VST 80_K2_AUTOV_CNR_V3
AND>(320) D4504 &0  ; VST 80_K2_AUTOV_CNR_V4
AND>(320) D4505 &0  ; VST 80_K2_AUTOV_CNR_V5
OUT 629.00  ; Autovask_K2_Hj1
LD TR0
ANDNOT 629.00  ; Autovask_K2_Hj1
OUT 1350.11  ; VST 80_K2_STARTIMPULS

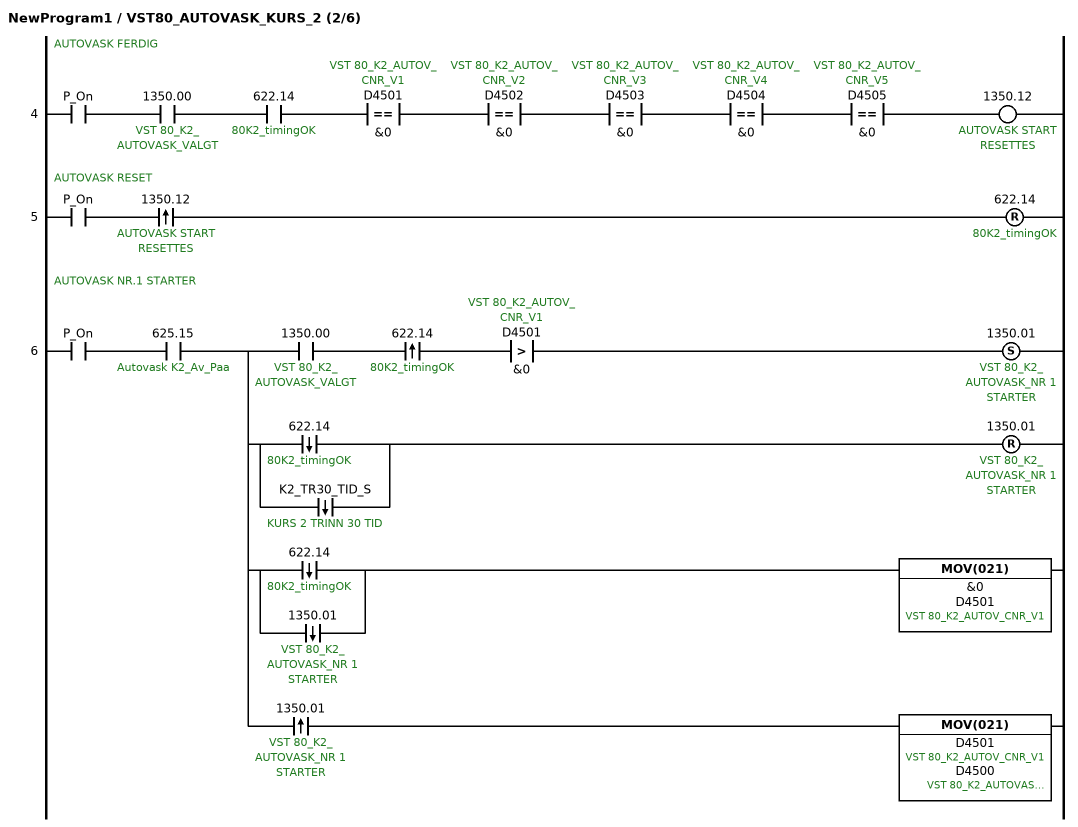
; rung 4: AUTOVASK FERDIG
LD P_On
AND 1350.00  ; VST 80_K2_AUTOVASK_VALGT
AND 622.14  ; 80K2_timingOK
AND=(300) D4501 &0  ; VST 80_K2_AUTOV_CNR_V1
AND=(300) D4502 &0  ; VST 80_K2_AUTOV_CNR_V2
AND=(300) D4503 &0  ; VST 80_K2_AUTOV_CNR_V3
AND=(300) D4504 &0  ; VST 80_K2_AUTOV_CNR_V4
AND=(300) D4505 &0  ; VST 80_K2_AUTOV_CNR_V5
OUT 1350.12  ; AUTOVASK START RESETTES
; rung 5: AUTOVASK RESET
LD P_On
@AND 1350.12  ; AUTOVASK START RESETTES
RSET 622.14  ; 80K2_timingOK
; rung 6: AUTOVASK NR.1 STARTER
LD P_On
AND 625.15  ; Autovask K2_Av_Paa
OUT TR0
AND 1350.00  ; VST 80_K2_AUTOVASK_VALGT
@AND 622.14  ; 80K2_timingOK
AND>(320) D4501 &0  ; VST 80_K2_AUTOV_CNR_V1
SET 1350.01  ; VST 80_K2_AUTOVASK_NR 1 STARTER
LD TR0
%LD 622.14  ; 80K2_timingOK
%OR K2_TR30_TID_S  ; KURS 2 TRINN 30 TID
ANDLD
RSET 1350.01  ; VST 80_K2_AUTOVASK_NR 1 STARTER
LD TR0
%LD 622.14  ; 80K2_timingOK
%OR 1350.01  ; VST 80_K2_AUTOVASK_NR 1 STARTER
ANDLD
MOV(021) &0 D4501  ; VST 80_K2_AUTOV_CNR_V1
LD TR0
@AND 1350.01  ; VST 80_K2_AUTOVASK_NR 1 STARTER
MOV(021) D4501 D4500  ; VST 80_K2_AUTOV_CNR_V1, VST 80_K2_AUTOVASK FELLESREGISTER

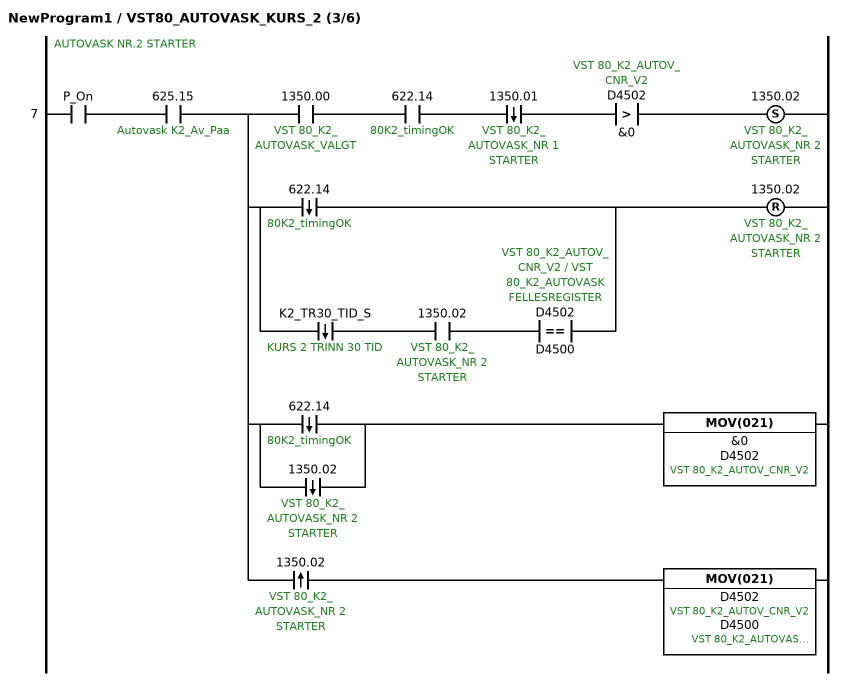
; rung 7: AUTOVASK NR.2 STARTER
LD P_On
AND 625.15  ; Autovask K2_Av_Paa
OUT TR0
AND 1350.00  ; VST 80_K2_AUTOVASK_VALGT
AND 622.14  ; 80K2_timingOK
%AND 1350.01  ; VST 80_K2_AUTOVASK_NR 1 STARTER
AND>(320) D4502 &0  ; VST 80_K2_AUTOV_CNR_V2
SET 1350.02  ; VST 80_K2_AUTOVASK_NR 2 STARTER
LD TR0
%LD 622.14  ; 80K2_timingOK
%LD K2_TR30_TID_S  ; KURS 2 TRINN 30 TID
AND 1350.02  ; VST 80_K2_AUTOVASK_NR 2 STARTER
AND=(300) D4502 D4500  ; VST 80_K2_AUTOV_CNR_V2, VST 80_K2_AUTOVASK FELLESREGISTER
ORLD
ANDLD
RSET 1350.02  ; VST 80_K2_AUTOVASK_NR 2 STARTER
LD TR0
%LD 622.14  ; 80K2_timingOK
%OR 1350.02  ; VST 80_K2_AUTOVASK_NR 2 STARTER
ANDLD
MOV(021) &0 D4502  ; VST 80_K2_AUTOV_CNR_V2
LD TR0
@AND 1350.02  ; VST 80_K2_AUTOVASK_NR 2 STARTER
MOV(021) D4502 D4500  ; VST 80_K2_AUTOV_CNR_V2, VST 80_K2_AUTOVASK FELLESREGISTER

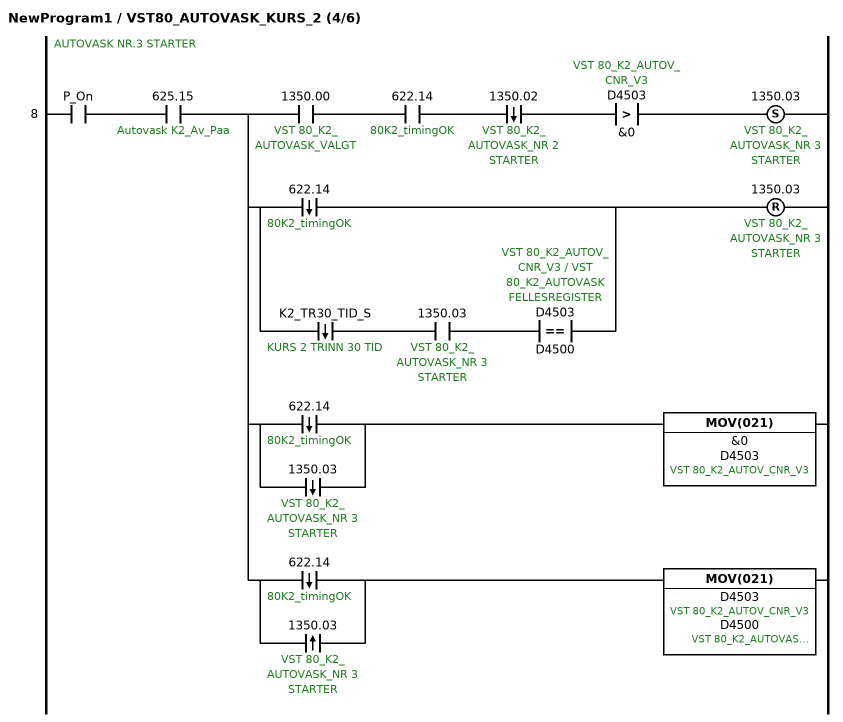
; rung 8: AUTOVASK NR.3 STARTER
LD P_On
AND 625.15  ; Autovask K2_Av_Paa
OUT TR0
AND 1350.00  ; VST 80_K2_AUTOVASK_VALGT
AND 622.14  ; 80K2_timingOK
%AND 1350.02  ; VST 80_K2_AUTOVASK_NR 2 STARTER
AND>(320) D4503 &0  ; VST 80_K2_AUTOV_CNR_V3
SET 1350.03  ; VST 80_K2_AUTOVASK_NR 3 STARTER
LD TR0
%LD 622.14  ; 80K2_timingOK
%LD K2_TR30_TID_S  ; KURS 2 TRINN 30 TID
AND 1350.03  ; VST 80_K2_AUTOVASK_NR 3 STARTER
AND=(300) D4503 D4500  ; VST 80_K2_AUTOV_CNR_V3, VST 80_K2_AUTOVASK FELLESREGISTER
ORLD
ANDLD
RSET 1350.03  ; VST 80_K2_AUTOVASK_NR 3 STARTER
LD TR0
%LD 622.14  ; 80K2_timingOK
%OR 1350.03  ; VST 80_K2_AUTOVASK_NR 3 STARTER
ANDLD
MOV(021) &0 D4503  ; VST 80_K2_AUTOV_CNR_V3
LD TR0
%LD 622.14  ; 80K2_timingOK
@OR 1350.03  ; VST 80_K2_AUTOVASK_NR 3 STARTER
ANDLD
MOV(021) D4503 D4500  ; VST 80_K2_AUTOV_CNR_V3, VST 80_K2_AUTOVASK FELLESREGISTER

